///Object base class for all classes
FUNCTION_BLOCK Object IMPLEMENTS IObject
VAR
    _className : STRING(50) := 'Object'; //Class name
    _version : STRING(8) := '1.0'; //Version
    firstPass : BOOL := FALSE; //First pass done
    _error : BOOL := FALSE; //Error
    _errorID : DWORD := 0; //Error id
    _errors : ErrorHistory; //Error history
END_VAR

///Add error to error history
METHOD PROTECTED AddError
VAR_INPUT
	errorID : DWORD; //Error ID
END_VAR
VAR
	addErrorLoop : INT;
END_VAR
FOR addErrorLoop := ObjectSetup.ErrorHistMax TO (ObjectSetup.ErrorHistMin + 1) BY -1 DO
	_errors[addErrorLoop] := _errors[addErrorLoop - 1];
END_FOR
_errors[ObjectSetup.ErrorHistMin] := errorID;
END_METHOD

(*Name, do not implement property override*)
PROPERTY ClassName : STRING(50)
GET
ClassName := _className;
END_GET
END_PROPERTY

///Control, override to get cyclic task in FB
METHOD INTERNAL Control
VAR_INPUT
END_VAR
END_METHOD

//Cycle Task, do not override this methode cyclic code is placed in M_Control 
METHOD FINAL CycleTask
IF NOT(firstPass) THEN
    firstPass := Init() = HResultSuccess.Done;
    IF NOT(firstPass) THEN
        RETURN;
	END_IF
END_IF
Control();
END_METHOD

(*Error, do not implement property override*)
PROPERTY Error : BOOL
GET
Error := _error;
END_GET
END_PROPERTY

(*error id, do not implement property override*)
PROPERTY ErrorID : DWORD
GET
ErrorID := _errorID;
END_GET
END_PROPERTY

(*Pointer to error history, do not implement property override*)
PROPERTY Errors : POINTER TO ErrorHistory
GET
Errors := ADR(_errors);
END_GET
END_PROPERTY

METHOD FB_init : BOOL
VAR_INPUT
	bInitRetains : BOOL; // if TRUE, the retain variables are initialized (warm start / cold start)
	bInCopyCode : BOOL;  // if TRUE, the instance afterwards gets moved into the copy code (online change)
END_VAR
firstPass := FALSE;
END_METHOD

///Initialize FB, Override to do custom initialize, no need to call super
METHOD INTERNAL Init : HRESULT
Init := HResultSuccess.Done;
END_METHOD

(*Reset error, allways call super*)
METHOD Reset
_error := FALSE;
_errorID := 0;
END_METHOD

///Set error on the Object and add entry to error history
METHOD PROTECTED SetError
VAR_INPUT
	errorID : DWORD; //Error ID
END_VAR
VAR
    setErrorLoop : INT;
END_VAR
IF NOT(_error) THEN
	_error := TRUE;
	THIS^._errorID := errorID;
	FOR setErrorLoop := ObjectSetup.ErrorHistMax TO (ObjectSetup.ErrorHistMin + 1) BY -1 DO
    	_errors[setErrorLoop] := _errors[setErrorLoop - 1];
	END_FOR
	_errors[ObjectSetup.ErrorHistMin] := _errorID;
END_IF
END_METHOD

(*Version,do not implement property override*)
PROPERTY Version : STRING(8)
GET
Version := _version;
END_GET
END_PROPERTY

END_FUNCTION_BLOCK

(* stored: Version 1.1.0.1, ProductVersion 3.1.4020.12
   POU Object: Id {7ae2b3bc-6889-427a-82e4-66c1a0f4f97f}, SpecialFunc None
   Method AddError: Id {26aececa-6134-4ea0-b147-75cddd786a49}
   Property ClassName: Id {e3a4abb1-c213-4331-ae82-93a6832e0b2b}
   Get Get: Id {360d13b5-cb0a-43c0-bb23-3319ceaa1789}
   Method Control: Id {b1c46935-f116-4df7-8461-83771a2e39a0}
   Method CycleTask: Id {eb714de1-926f-48dc-8981-1ce3b30d9fbe}
   Property Error: Id {d41bc890-e3af-4a7c-8e60-f03a1c619e63}
   Get Get: Id {adec9c0c-9263-40fa-8b89-e0381541d2fc}
   Property ErrorID: Id {63ffb5b2-2ae5-4a47-86b8-36564ac6ed39}
   Get Get: Id {2ddbd3ca-8dd1-411b-b481-2e4f78bb8567}
   Property Errors: Id {fcbaa8a8-a2ef-4477-8ff4-d26aef6ce2a5}
   Get Get: Id {166ae521-9fb5-47c9-a237-1559e097c4e2}
   Method FB_init: Id {3ab89805-0d3a-421a-8ebd-105e5791755c}
   Method Init: Id {4237cb80-d346-4a7c-938a-6d6c8c793f75}
   Method Reset: Id {9560225a-1cab-4c8f-9ae8-4c6933de2dbc}
   Method SetError: Id {f7b289ae-e020-441f-a57b-6988eb02710a}
   Property Version: Id {41ae7693-4c80-4a34-85a8-401771f8ba14}
   Get Get: Id {0e91d3fe-1da8-4005-902d-a36628829292} *)
